Program P30_ManualControlExt
VAR
	analogDeviceRampControl : FB_AnalogDeviceRampControl;
END_VAR

analogDeviceRampControl();

END_PROGRAM

(* stored: Version 1.1.0.1, ProductVersion 3.1.4026.11
   POU P30_ManualControlExt: Id {87edd900-96de-41d7-b820-4b4e090513ec}, SpecialFunc None *)
